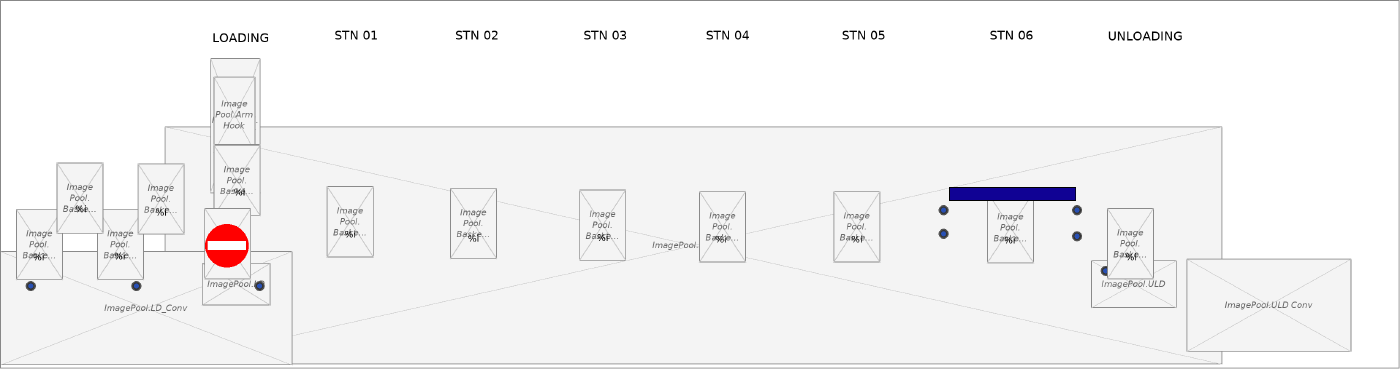
VISUALIZATION Popup_Machine  // 1658x438
    Rectangle (0,0 1658x438)
    Image (195,150 1252x282), image: ImagePool.Machine
    Label (379,22 86x40), "STN 01"
    Label (522,22 86x40), "STN 02"
    Label (674,22 86x40), "STN 03"
    Label (819,22 86x40), "STN 04"
    Label (980,22 86x40), "STN 05"
    Label (1155,22 86x40), "STN 06"
    Label (232,22 106x46), "LOADING"
    Label (1294,22 125x42), "UNLOADING"
    Image (0,298 346x135), image: ImagePool.LD_Conv
    Image (239,312 81x50), image: ImagePool.LD
    Image (249,69 59x160), image: ImagePool.Arm Body
        p3560616238: HMI_Function.MotionX
    Image (253,91 49x90), image: ImagePool.Arm Hook
        p3560616238: HMI_Function.MotionX
        p2738717112: HMI_Function.MotionY
    Image (1405,307 195x110), image: ImagePool.ULD Conv
    Image (1292,309 101x56), image: ImagePool.ULD
    Lamp1 (301,333 13x13), variable: ARbDI[eX13002_LoadingConveyorSensor_Pick], style: Lamp-Lamp1-Blue
    Lamp1 (1303,315 13x13), variable: ARbDI[eX12011_UnloadingSensor_BasketDetection], style: Lamp-Lamp1-Blue
    Image (387,221 55x84), invisible if: NOT.ARbBasketBdFlag[2], image: ImagePool.Basket Red
    Rectangle (399,261 32x31), "%i", text variable: DSStnBasketInfo[1].iProductRecipeNo, invisible if: NOT.ARbBasketBdFlag[2]
    Group (387,221 55x84)
        Image (0,0 55x84), invisible if: NOT.ARbBasketGdFlag[2], image: ImagePool.Basket Green
        Rectangle (12,42 32x31), "%i", text variable: DSStnBasketInfo[1].iProductRecipeNo, invisible if: NOT.ARbBasketGdFlag[2]
    Group (533,223 55x84)
        Image (0,0 55x84), invisible if: NOT.ARbBasketBdFlag[3], image: ImagePool.Basket Red
        Rectangle (11,44 32x31), "%i", text variable: DSStnBasketInfo[2].iProductRecipeNo, invisible if: NOT.ARbBasketBdFlag[3]
    Group (533,223 55x84)
        Image (0,0 55x84), invisible if: NOT.ARbBasketGdFlag[3], image: ImagePool.Basket Green
        Rectangle (12,45 32x31), "%i", text variable: DSStnBasketInfo[2].iProductRecipeNo, invisible if: NOT.ARbBasketGdFlag[3]
    Image (686,225 55x84), invisible if: NOT.ARbBasketBdFlag[4], image: ImagePool.Basket Red
    Rectangle (698,268 32x31), "%i", text variable: DSStnBasketInfo[3].iProductRecipeNo, invisible if: NOT.ARbBasketBdFlag[4]
    Group (686,225 55x84)
        Image (0,0 55x84), invisible if: NOT.ARbBasketGdFlag[4], image: ImagePool.Basket Green
        Rectangle (12,42 32x31), "%i", text variable: DSStnBasketInfo[3].iProductRecipeNo, invisible if: NOT.ARbBasketGdFlag[4]
    Group (828,227 55x84)
        Image (0,0 55x84), invisible if: NOT.ARbBasketBdFlag[5], image: ImagePool.Basket Red
        Rectangle (12,43 32x31), "%i", text variable: DSStnBasketInfo[4].iProductRecipeNo, invisible if: NOT.ARbBasketBdFlag[5]
    Group (828,227 55x84)
        Image (0,0 55x84), invisible if: NOT.ARbBasketGdFlag[5], image: ImagePool.Basket Green
        Rectangle (10,42 32x31), "%i", text variable: DSStnBasketInfo[4].iProductRecipeNo, invisible if: NOT.ARbBasketGdFlag[5]
    Group (987,227 55x84)
        Image (0,0 55x84), invisible if: NOT.ARbBasketBdFlag[6], image: ImagePool.Basket Red
        Rectangle (12,43 32x31), "%i", text variable: DSStnBasketInfo[5].iProductRecipeNo, invisible if: NOT.ARbBasketBdFlag[6]
    Group (987,227 55x84)
        Image (0,0 55x84), invisible if: NOT.ARbBasketGdFlag[6], image: ImagePool.Basket Green
        Rectangle (12,42 32x31), "%i", text variable: DSStnBasketInfo[5].iProductRecipeNo, invisible if: NOT.ARbBasketGdFlag[6]
    Group (1169,228 55x84)
        Image (0,0 55x84), invisible if: NOT.ARbBasketBdFlag[7], image: ImagePool.Basket Red
        Rectangle (13,42 32x31), "%i", text variable: DSStnBasketInfo[6].iProductRecipeNo, invisible if: NOT.ARbBasketBdFlag[7]
    Group (1169,228 55x84)
        Image (0,0 55x84), invisible if: NOT.ARbBasketGdFlag[7], image: ImagePool.Basket Green
        Rectangle (11,42 32x31), "%i", text variable: DSStnBasketInfo[6].iProductRecipeNo, invisible if: NOT.ARbBasketGdFlag[7]
    Group (1311,247 55x84)
        Image (0,0 55x84), invisible if: NOT.ARbBasketBdFlag[12], image: ImagePool.Basket Red
        Rectangle (12,42 32x31), "%i", text variable: AR2sDSCv_UldConfirmBasketInfo[1,1].iProductRecipeNo, invisible if: NOT.ARbBasketBdFlag[12]
    Group (1311,247 55x84)
        Image (0,0 55x84), invisible if: NOT.ARbBasketGdFlag[12], image: ImagePool.Basket Green
        Rectangle (13,43 32x31), "%i", text variable: AR2sDSCv_UldConfirmBasketInfo[1,1].iProductRecipeNo, invisible if: NOT.ARbBasketGdFlag[12]
    Image (253,171 55x84), invisible if: NOT.ARbBasketBdFlag[16], image: ImagePool.Basket Red
        p2738717112: HMI_Function.MotionY
        p3560616238: HMI_Function.MotionX
    Rectangle (269,214 32x31), "%i", text variable: DSArmBasketInfo[1].iProductRecipeNo, invisible if: NOT.ARbBasketBdFlag[16]
        p3560616238: HMI_Function.MotionX
        p2738717112: HMI_Function.MotionY
    Image (253,172 55x84), invisible if: NOT.ARbBasketGdFlag[16], image: ImagePool.Basket Green
        p3560616238: HMI_Function.MotionX
        p2738717112: HMI_Function.MotionY
    Rectangle (268,213 32x31), "%i", text variable: DSArmBasketInfo[1].iProductRecipeNo, invisible if: NOT.ARbBasketGdFlag[16]
        p3560616238: HMI_Function.MotionX
        p2738717112: HMI_Function.MotionY
    Group (242,247 55x84)
        Image (0,0 55x84), invisible if: NOT.ARbBasketGdFlag[1], image: ImagePool.Basket Green
        Rectangle (10,42 32x31), "%i", text variable: AR2sDSCv_LdConfirmBasketInfo[1,3].iProductRecipeNo, invisible if: NOT.ARbBasketGdFlag[1]
    Group (115,248 55x84)
        Image (0,0 55x84), invisible if: NOT AR2sDSCv_LdConfirmBasketInfo[1,2].bAvailibility, image: ImagePool.Basket Green
        Rectangle (11,41 32x31), "%i", text variable: AR2sDSCv_LdConfirmBasketInfo[1,2].iProductRecipeNo, invisible if: NOT AR2sDSCv_LdConfirmBasketInfo[1,2].bAvailibility
    Group (19,248 55x84)
        Image (0,0 55x84), invisible if: NOT AR2sDSCv_LdConfirmBasketInfo[1,1].bAvailibility, image: ImagePool.Basket Green
        Rectangle (11,42 32x31), "%i", text variable: AR2sDSCv_LdConfirmBasketInfo[1,1].iProductRecipeNo, invisible if: NOT AR2sDSCv_LdConfirmBasketInfo[1,1].bAvailibility
    Group (67,193 55x84)
        Image (0,0 55x84), invisible if: NOT AR2sDSCv_LdTransferBasketInfo[1,1].bAvailibility, image: ImagePool.Basket Blue
        Rectangle (13,40 32x31), "%i", text variable: AR2sDSCv_LdTransferBasketInfo[1,1].iProductRecipeNo, invisible if: NOT AR2sDSCv_LdTransferBasketInfo[1,1].bAvailibility
    Group (163,194 55x84)
        Image (0,0 55x84), invisible if: NOT AR2sDSCv_LdTransferBasketInfo[1,2].bAvailibility, image: ImagePool.Basket Blue
        Rectangle (12,43 32x31), "%i", text variable: AR2sDSCv_LdTransferBasketInfo[1,2].iProductRecipeNo, invisible if: NOT AR2sDSCv_LdTransferBasketInfo[1,2].bAvailibility
    Group (243,266 51x51), invisible if: NOT bBlockBasketEnter
        Ellipse (0,0 51x51)
        Rectangle (3,20 45x10)
    Lamp1 (30,333 13x13), variable: ARbDI[eX13000_LoadingConveyorSensor_Feed], style: Lamp-Lamp1-Blue
    Lamp1 (155,333 13x13), variable: ARbDI[eX13001_LoadingConveyorSensor_Index], style: Lamp-Lamp1-Blue
    Lamp1 (1111,243 13x13), variable: ARbDI[eX12101_Stn06SlidingDoorRs01_Unclamp], style: Lamp-Lamp1-Blue
    Lamp1 (1111,271 13x13), variable: ARbDI[eX12100_Stn06SlidingDoorRs01_Clamp], style: Lamp-Lamp1-Blue
    Lamp1 (1269,274 13x13), variable: ARbDI[eX12102_Stn06SlidingDoorRs02_Clamp], style: Lamp-Lamp1-Blue
    Lamp1 (1269,243 13x13), variable: ARbDI[eX12103_Stn06SlidingDoorRs02_Unclamp], style: Lamp-Lamp1-Blue
    Rectangle (1124,222 150x16), invisible if: NOT ARbDI[eX12008_Stn06SlidingDoorRs_Close]
END_VISUALIZATION

(* stored: Version 1.1.0.1, ProductVersion 3.1.4024.12
   Visu Popup_Machine: Id {5de16b85-3394-4b76-9857-58513c54f52c} *)
